FUNCTION fuzzyAND : REAL
VAR_INPUT
	ANDmethod:eAndMethod;
	in1,in2:REAL;
END_VAR

CASE ANDmethod OF
	eAndMethod.Minimum://***********
		fuzzyAND := MIN(in1,in2);
	eAndMethod.Product://***********
		fuzzyAND := in1*in2;
END_CASE

END_FUNCTION

(* stored: Version 1.1.0.1, ProductVersion 3.1.4024.6
   POU fuzzyAND: Id {e5edcf6b-2f4e-4d5f-a4f1-49acc34c49ab}, SpecialFunc None *)
